{attribute 'GeneratedUsingTerminal: AT2040-0250-0024'}
{attribute addProperty BoxType "AT2040-0250-0024"}
{attribute addProperty Id "A_0105_AT2026_5250_0018_AT2026_5250AT2026_01D6DEDF80"}
{attribute addProperty CRC "2781264902"}
{attribute addProperty Size "80"}
TYPE A_0039_AT2040_0250_0024_A5C6BC06 EXTENDS AT2040_86175B41 :
STRUCT
	{attribute addProperty Name "A_0105_AT2026_5250_0018_AT2026_5250"}
	A_0105_AT2026_5250_0018_AT2026_5250 : AT2026_01D6DEDF;
END_STRUCT
END_TYPE

(* stored: Version 1.2.0.0, ProductVersion 3.1.4024.9
   DUT A_0039_AT2040_0250_0024_A5C6BC06: Id {0e85b859-b79a-449c-b676-4a6600dd4603} *)
